Staubli VAL3: oFluorDet.pgx

public program oFluorDet(num nChoice (dimensions=1))
// oFluorDet
begin
  dioSet(oFluorDet,nChoice)
end
